FUNCTION_BLOCK TEST_GEN (* Test GE functions of numerical values *)
  (* Standard: IEC 61499-1 *)
  (* Version 0.0, 2006-09-11, JHC, Holobloc Inc *)
  (* Compiler header: package fb.rt.test; *)
  (* Compiler classdef: SimpleFB *)
  (* Compiler Java Sun JDK 1.5.0 *)
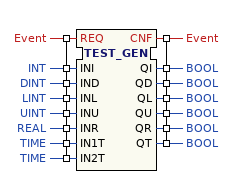
  EVENT_INPUT
    REQ WITH INI, INL, INU, IND, INR, IN1T, IN2T;
  END_EVENT
  EVENT_OUTPUT
    CNF WITH QI, QD, QL, QU, QR, QT;
  END_EVENT
  VAR_INPUT
    INI : INT;
    IND : DINT;
    INL : LINT;
    INU : UINT;
    INR : REAL;
    IN1T : TIME;
    IN2T : TIME;
  END_VAR
  VAR_OUTPUT
    QI : BOOL;
    QD : BOOL;
    QL : BOOL;
    QU : BOOL;
    QR : BOOL;
    QT : BOOL;
  END_VAR
  ALGORITHM REQ IN FBD:
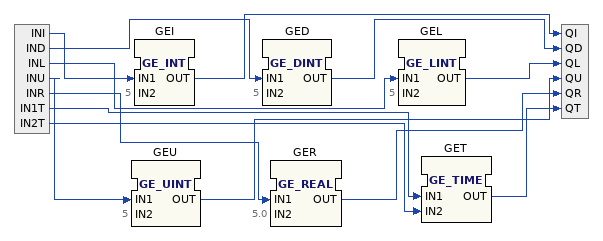
    FBS
      GEI : GE_INT(IN2 := 5);
      GED : GE_DINT(IN2 := 5);
      GEL : GE_LINT(IN2 := 5);
      GEU : GE_UINT(IN2 := 5);
      GER : GE_REAL(IN2 := 5.0);
      GET : GE_TIME;
    END_FBS
    DATA_CONNECTIONS
      INI TO GEI.IN1;
      IND TO GED.IN1;
      INL TO GEL.IN1;
      INU TO GEU.IN1;
      INR TO GER.IN1;
      GEI.OUT TO QI;
      GED.OUT TO QD;
      GEL.OUT TO QL;
      GEU.OUT TO QU;
      GER.OUT TO QR;
      GET.OUT TO QT;
      IN1T TO GET.IN1;
      IN2T TO GET.IN2;
    END_CONNECTIONS
  END_ALGORITHM
END_FUNCTION_BLOCK
